{attribute 'qualified_only'}
{attribute 'strict'}
TYPE TrajectoryState :
(
  Undefined,
  Idle,
  Busy,
  Error
);
END_TYPE

(* stored: Version 1.1.0.1
   DUT TrajectoryState: Id {1b401aa7-ce7a-4de0-8dde-e86175fd1d75} *)
